INTERFACE I_VisitModules

METHOD VisitModule
VAR_INPUT
	Module : I_Module;
END_VAR
END_METHOD

END_INTERFACE

(* stored: Version 1.1.0.1, ProductVersion 3.1.4024.12
   Itf I_VisitModules: Id {a1a9879c-aa7b-4caa-8103-ae67298d8601}
   Method VisitModule: Id {a6787921-a92b-4aee-9d38-2c80c40710b5} *)
